FUNCTION_BLOCK PID_Regler
VAR_INPUT
	ref : REAL;						// Aktuelle Referenzgrösse (Soll-Grösse)
 	y : REAL;						// Aktuelle Regelgrösse (Ist-Grösse)
	Modus : System_Modus_Enum;		// Aktueller Modus (Init oder Run)
	Param : PID_Parameter_Strukt;	// Parameter der PID Reglers
	T : REAL;						// Abtastzeit
END_VAR
VAR_OUTPUT
	u_r : REAL;						// Stellgrösse Output
END_VAR
VAR
	u_k: REAL;						// P-Anteil des Reglers
	u_i_k: REAL;					// I-Anteil des Reglers
	u_d_k: REAL;					// D-Anteil des Reglers
	
	u_i_k_1: REAL;					// I-Anteil u_i[k-1]
	
	e_k: REAL;						// Fehler e_k := ref - y;
	e_k_1: REAL;					// Fehler e[k-1]
	
	i: REAL;						// Param.K_p / Param.T_i i-Faktor
	ad: REAL;						// Vorfaktor D-Anteil
	bd: REAL;						// Vorfaktor D-Anteil
	u_d_k_1: REAL;					// D-Anteil u_d[k-1]
	u_r_oS: REAL;					// u_r ohne Sättigung
	y_1: REAL;
END_VAR

// Repräsentiert den Regler

// CPU Belastung minimieren und soviel wie möglich schon im Init Modus berechnen
CASE Modus OF
	/// UNDEFINED ////
	System_Modus_Enum.enum_member:
		Modus := System_Modus_Enum.System_Init;
	
	/// INIT ///
	System_Modus_Enum.System_Init:
		i := Param.K_p / Param.T_i;
		Param.N := 20;
		ad := Param.T_d / (Param.T_d + Param.N * T);
		bd := (Param.K_p * Param.N * Param.T_d) / (Param.T_d + Param.N * T);
		Param.Tr := 0.003162;
	
	/// RUN ///
	System_Modus_Enum.System_Run:
		e_k := ref - y;
		// A4: Diskretisiere den P-Anteil des analogen PID Reglers
		// Gibt keine andere Möglichkeit für u_k
		
		// P-Anteil
		u_k := Param.K_p * e_k;
		
		// A6: D-Anteil mit der Rückwärtsrechteckregel
		u_d_k :=  (ad * u_d_k_1 + bd * (e_k - e_k_1));
		
		// Ohne Sättigung
		u_r_oS := u_k + u_i_k + u_d_k;
		
		// AS_8_A_1 Mit Saturation
		IF u_r_oS > param.u_max THEN
			u_r := Param.u_max;
		ELSIF u_r_oS < param.u_min THEN
			u_r := Param.u_min;
		ELSE
			// Sättigungsbereich nicht Erreicht und somit einfache Zuweisung
			u_r := u_r_oS;
		END_IF
		
		// Anti Reset (ARW) AS_8
		IF Param.ARW THEN
			// Mit Anti-Reset Windup. I-Anteil limitieren
			u_i_k := u_i_k_1 + i * ((e_k + e_k_1) / 2) * T + (T / Param.Tr) * (u_r - u_r_oS);
		ELSE
			// A5: Diskretisiere den I-Anteil des analogen PID Reglers mit Trapezregel (in Rek. Form)
			u_i_k := u_i_k_1 + i * ((e_k + e_k_1) / 2) * T;
		END_IF
		
		
		// Zuweisung alter Werte
		e_k_1 := e_k;
		u_d_k_1 := u_d_k;
		u_i_k_1 := u_i_k;
		y_1 := y;
		
	
END_CASE

END_FUNCTION_BLOCK

(* stored: Version 1.1.0.1, ProductVersion 3.1.4024.9
   POU PID_Regler: Id {7dcd331b-5f89-4474-abe4-edc66f385524}, SpecialFunc None *)
